// TIA Portal V20 export
// export: Created 2025-12-01T14:57:41.1647869Z, ExportSetting None, DisplayName Totally Integrated Automation Portal, DisplayVersion V20 Update 3, DisplayName TIA Portal Openness, DisplayVersion V20 Update 3, DisplayName TIA Portal Version Control Interface, DisplayVersion V20 Update 3, DisplayName STEP 7 Professional, DisplayVersion V20 Update 3, DisplayName STEP 7 Safety, DisplayVersion V20 Update 2, DisplayName WinCC Basic/Comfort/Advanced, DisplayVersion V20 Update 3, DisplayName WinCC Professional, DisplayVersion V20 Update 3, DisplayName WinCC Unified, DisplayVersion V20 Update 3
FUNCTION_BLOCK "FB384_Enfardadora_Paletizador_NDD"   // FB384, LAD
{ S7_Optimized_Access := 'FALSE' }
// stored: AutoNumber false, SetENOAutomatically false
   VAR_INPUT
      EstadoZona : "EstadoZona";
      NDB_Enfardadora : UInt;
      NumMaquina : UInt;
      PosicionActual : Int;
      DesHabitar_Enfa : Bool;
      PorCapas_Enfa : Bool;
      CheckElev_EnEnfardadora : Bool;
   END_VAR
   VAR
      MemoPosicionActual : Int;
      PosicionEnfardado : Int;
      VelocidadEnfardado : Int;
      ProgramaEnfardado : Int;
      PosEnfardadora_OK : Bool;
      PeticionSubirELEV : Bool;
      PeticionBajarELEV : Bool;
      EnPosEnfardado : Bool;
      DebajoPosEnfardado : Bool;
      EnPaletizadoUT : Bool;
      FinPaletizadoUT : Bool;
      SinEnfardadoUT { ExternalVisible := 'False'} : Bool;
      ConEnfardadoUT { ExternalVisible := 'False'} : Bool;
      IniciarEnfardado : Bool;
      FinEnfardado : Bool;
      ErrorEnfardado : Bool;
      RealizaCapaUT : Bool;
      HaciendoCapas : Bool;
      EnCicloEnfardado : Bool;
      EnCicloCapas : Bool;
      Elev_Subiendo : Bool;
      Elev_Bajando : Bool;
      ENFA_ET00 : Bool;
      ENFA_ET01 : Bool;
      ENFA_ET10 : Bool;
      ENFA_ET11 : Bool;
      ENFA_ET20 : Bool;
      ENFA_ET21 : Bool;
      ENFA_ET02 : Bool;
      ENFA_ET50 : Bool;
      ENFA_ET51 { ExternalVisible := 'False'} : Bool;
      t_march_enfa { S7_SetPoint := 'True'} : CTD_INT;
   END_VAR
   VAR_TEMP
      Entradas : "NDD_Enfardadora_Input";
      Salidas : "NDD_Enfardadora_Output";
      Guardar_AR1 : DWord;
      Guardar_AR2 : DWord;
      DB_Enfardadora : Word;
      P_Entradas : DWord;
      P_Salidas : DWord;
      P_Temporal : DWord;
      Margen : Int;
      AuxPosMax : Int;
      AuxPosMin : Int;
      Maquina : Word;
      DB_ColasMesas : Word;
      DB_DatosUT : Word;
      NumeroUT : UInt;
      SiguienteUT : UInt;
      MesaActual : UInt;
      MesaDestino : UInt;
      SinUT : Bool;
      AuxEstados : Bool;
   END_VAR
BEGIN

REGION Network 1: Inicializacion
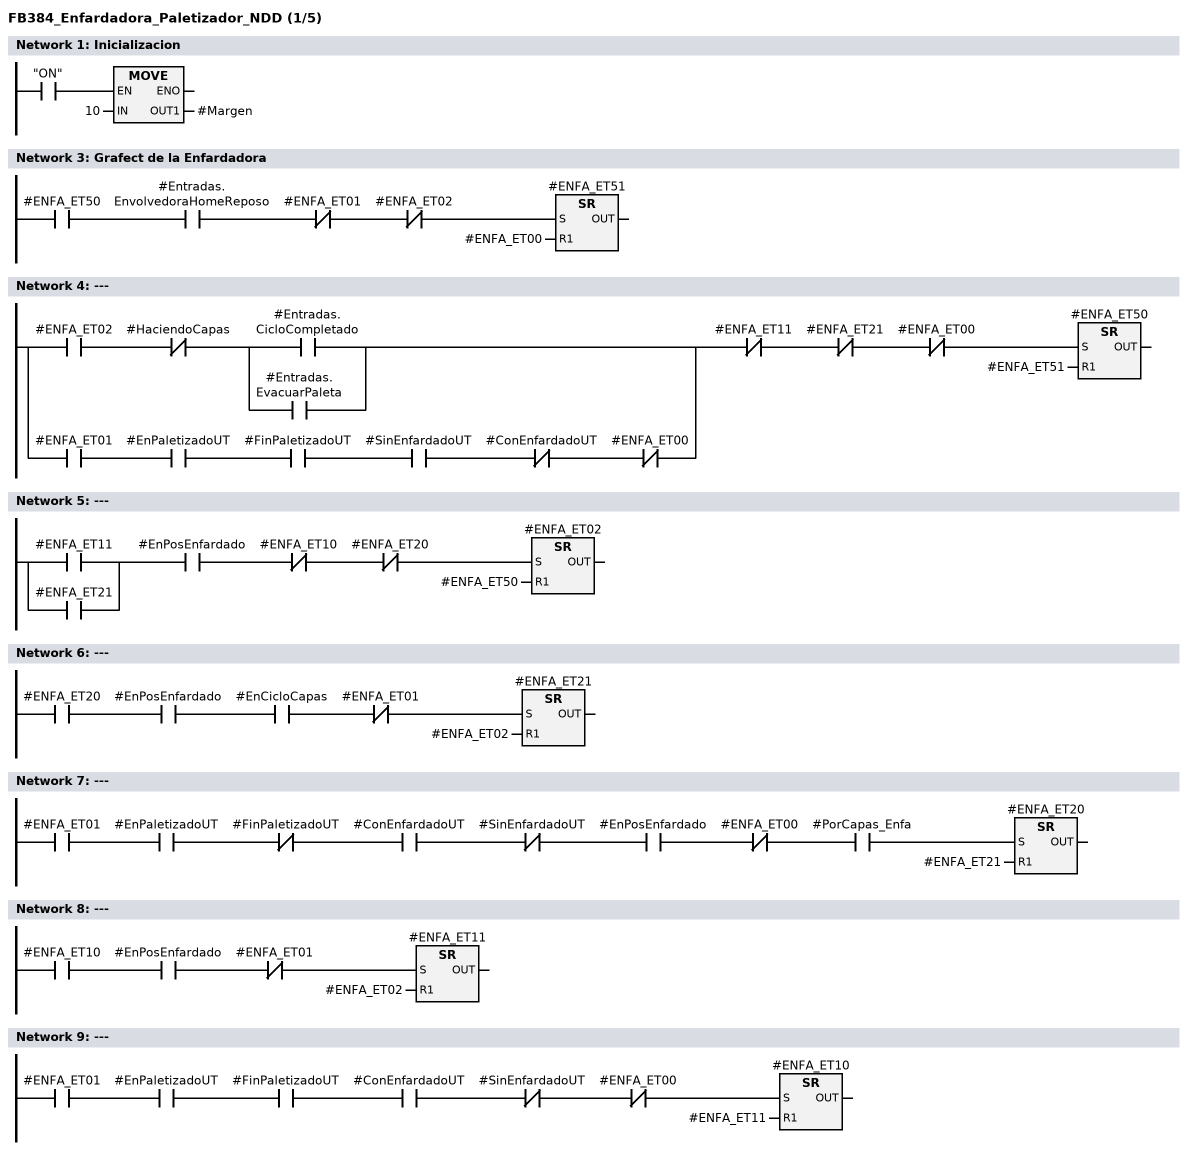
   RUNG wire#powerrail
      Contact( "ON" )
      { S7_GenerateENO := "TRUE" } Move(in := 10, out1 => #Margen)
   END_RUNG
   // the same network as SCL:
   IF "ON" THEN #Margen := 10; END_IF;
END_REGION

NETWORK
TITLE = Lectura de Datos
/////////////////////////////////////////////////////////////////////
/////////////////////////////////////////////////////////////////////
// - Inicializaciones Previas

      TAR1  #Guardar_AR1;  // - Guardar el AR1

      L     #NumMaquina;  // - Numero de Maquina
      T     #Maquina;

      L     #NDB_Enfardadora;  // - Numero de DB de Interlock
      T     #DB_Enfardadora;

/////////////////////////////////////////////////////////////////////
// -- Leer las entradas y salidas de la Enfardadora

      L     P##Entradas;  // --- Leer las Entradas
      T     #P_Entradas;
      L     P#0.0;
      T     #P_Temporal;

      OPN   DB [#DB_Enfardadora];  // - Bits de la Enfardadora
      L     DBD [#P_Temporal];
      T     LD [#P_Entradas];

      L     P#4.0;
      T     #P_Temporal;
      OPN   DB [#DB_Enfardadora];  // - Velocidad de Enfaradado
      L     DBW [#P_Temporal];
      T     #Entradas.VelocidadElevador;

      L     P#6.0;
      T     #P_Temporal;
      OPN   DB [#DB_Enfardadora];  // - Altura de Inicio de Enfardado
      L     DBW [#P_Temporal];
      T     #Entradas.AlturaInicioEnfardado;

      L     0;
      T     #Entradas.Libre_Int_08;

      L     P##Salidas;  // --- Leer las Salidas
      T     #P_Salidas;
      L     P#10.0;
      T     #P_Temporal;

      OPN   DB [#DB_Enfardadora];  // --- Bits
      L     DBD [#P_Temporal];
      T     LD [#P_Salidas];

      L     P#14.0;
      T     #P_Temporal;
      OPN   DB [#DB_Enfardadora];  // - Altura de la Paleta
      L     DBW [#P_Temporal];
      T     #Salidas.AlturaPaleta;

      L     P#16.0;
      T     #P_Temporal;
      OPN   DB [#DB_Enfardadora];  // - Posicion del Elevador
      L     DBW [#P_Temporal];
      T     #Salidas.AlturaElevador;

      L     P#18.0;
      T     #P_Temporal;
      OPN   DB [#DB_Enfardadora];  // - Programa
      L     DBW [#P_Temporal];
      T     #Salidas.Programa;


/////////////////////////////////////////////////////////////////////
/////////////////////////////////////////////////////////////////////
//  - Finalizacion

      LAR1  #Guardar_AR1;  // - Recuperar el AR1



REGION Network 3: Grafect de la Enfardadora
   RUNG wire#powerrail
      Contact( #ENFA_ET50 )
      Contact( #Entradas.EnvolvedoraHomeReposo )
      I_Contact( #ENFA_ET01 )
      I_Contact( #ENFA_ET02 )
      S_SR(operand := #ENFA_ET51, r1 := #ENFA_ET00)
   END_RUNG
   // the same network as SCL:
   IF #ENFA_ET50 AND #Entradas.EnvolvedoraHomeReposo AND NOT #ENFA_ET01 AND NOT #ENFA_ET02 THEN
       #ENFA_ET51 := TRUE;   // SR flip-flop
   END_IF;
   IF #ENFA_ET00 THEN #ENFA_ET51 := FALSE; END_IF;
END_REGION

REGION Network 4: ---
   RUNG wire#powerrail
      Contact( #ENFA_ET02 )
      I_Contact( #HaciendoCapas )
      wire#w1
      Contact( #Entradas.CicloCompletado )
      wire#w2
      I_Contact( #ENFA_ET11 )
      I_Contact( #ENFA_ET21 )
      I_Contact( #ENFA_ET00 )
      S_SR(operand := #ENFA_ET50, r1 := #ENFA_ET51)
   END_RUNG
   RUNG wire#w1
      Contact( #Entradas.EvacuarPaleta )
   END_RUNG wire#w2
   RUNG wire#powerrail
      Contact( #ENFA_ET01 )
      Contact( #EnPaletizadoUT )
      Contact( #FinPaletizadoUT )
      Contact( #SinEnfardadoUT )
      I_Contact( #ConEnfardadoUT )
      I_Contact( #ENFA_ET00 )
   END_RUNG wire#w2
   // the same network as SCL:
   IF ((#ENFA_ET02 AND NOT #HaciendoCapas AND (#Entradas.CicloCompletado OR #Entradas.EvacuarPaleta)) OR (#ENFA_ET01 AND #EnPaletizadoUT AND #FinPaletizadoUT AND #SinEnfardadoUT AND NOT #ConEnfardadoUT AND NOT #ENFA_ET00)) AND NOT #ENFA_ET11 AND NOT #ENFA_ET21 AND NOT #ENFA_ET00 THEN
       #ENFA_ET50 := TRUE;   // SR flip-flop
   END_IF;
   IF #ENFA_ET51 THEN #ENFA_ET50 := FALSE; END_IF;
END_REGION

REGION Network 5: ---
   RUNG wire#powerrail
      Contact( #ENFA_ET11 )
      wire#w1
      Contact( #EnPosEnfardado )
      I_Contact( #ENFA_ET10 )
      I_Contact( #ENFA_ET20 )
      S_SR(operand := #ENFA_ET02, r1 := #ENFA_ET50)
   END_RUNG
   RUNG wire#powerrail
      Contact( #ENFA_ET21 )
   END_RUNG wire#w1
   // the same network as SCL:
   IF (#ENFA_ET11 OR #ENFA_ET21) AND #EnPosEnfardado AND NOT #ENFA_ET10 AND NOT #ENFA_ET20 THEN
       #ENFA_ET02 := TRUE;   // SR flip-flop
   END_IF;
   IF #ENFA_ET50 THEN #ENFA_ET02 := FALSE; END_IF;
END_REGION

REGION Network 6: ---
   RUNG wire#powerrail
      Contact( #ENFA_ET20 )
      Contact( #EnPosEnfardado )
      Contact( #EnCicloCapas )
      I_Contact( #ENFA_ET01 )
      S_SR(operand := #ENFA_ET21, r1 := #ENFA_ET02)
   END_RUNG
   // the same network as SCL:
   IF #ENFA_ET20 AND #EnPosEnfardado AND #EnCicloCapas AND NOT #ENFA_ET01 THEN
       #ENFA_ET21 := TRUE;   // SR flip-flop
   END_IF;
   IF #ENFA_ET02 THEN #ENFA_ET21 := FALSE; END_IF;
END_REGION

REGION Network 7: ---
   RUNG wire#powerrail
      Contact( #ENFA_ET01 )
      Contact( #EnPaletizadoUT )
      I_Contact( #FinPaletizadoUT )
      Contact( #ConEnfardadoUT )
      I_Contact( #SinEnfardadoUT )
      Contact( #EnPosEnfardado )
      I_Contact( #ENFA_ET00 )
      Contact( #PorCapas_Enfa )
      S_SR(operand := #ENFA_ET20, r1 := #ENFA_ET21)
   END_RUNG
   // the same network as SCL:
   IF #ENFA_ET01 AND #EnPaletizadoUT AND NOT #FinPaletizadoUT AND #ConEnfardadoUT AND NOT #SinEnfardadoUT AND #EnPosEnfardado AND NOT #ENFA_ET00 AND #PorCapas_Enfa THEN
       #ENFA_ET20 := TRUE;   // SR flip-flop
   END_IF;
   IF #ENFA_ET21 THEN #ENFA_ET20 := FALSE; END_IF;
END_REGION

REGION Network 8: ---
   RUNG wire#powerrail
      Contact( #ENFA_ET10 )
      Contact( #EnPosEnfardado )
      I_Contact( #ENFA_ET01 )
      S_SR(operand := #ENFA_ET11, r1 := #ENFA_ET02)
   END_RUNG
   // the same network as SCL:
   IF #ENFA_ET10 AND #EnPosEnfardado AND NOT #ENFA_ET01 THEN
       #ENFA_ET11 := TRUE;   // SR flip-flop
   END_IF;
   IF #ENFA_ET02 THEN #ENFA_ET11 := FALSE; END_IF;
END_REGION

REGION Network 9: ---
   RUNG wire#powerrail
      Contact( #ENFA_ET01 )
      Contact( #EnPaletizadoUT )
      Contact( #FinPaletizadoUT )
      Contact( #ConEnfardadoUT )
      I_Contact( #SinEnfardadoUT )
      I_Contact( #ENFA_ET00 )
      S_SR(operand := #ENFA_ET10, r1 := #ENFA_ET11)
   END_RUNG
   // the same network as SCL:
   IF #ENFA_ET01 AND #EnPaletizadoUT AND #FinPaletizadoUT AND #ConEnfardadoUT AND NOT #SinEnfardadoUT AND NOT #ENFA_ET00 THEN
       #ENFA_ET10 := TRUE;   // SR flip-flop
   END_IF;
   IF #ENFA_ET11 THEN #ENFA_ET10 := FALSE; END_IF;
END_REGION

REGION Network 10: ---
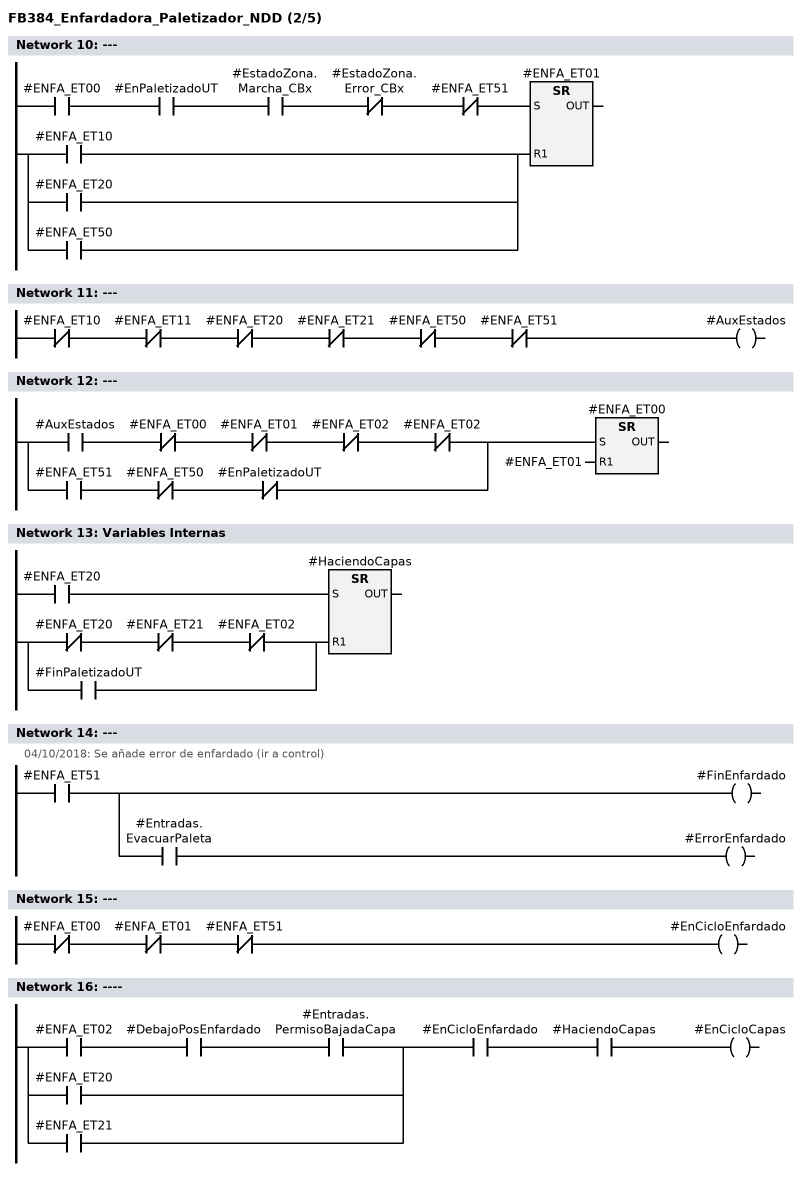
   RUNG wire#powerrail
      Contact( #ENFA_ET00 )
      Contact( #EnPaletizadoUT )
      Contact( #EstadoZona.Marcha_CBx )
      I_Contact( #EstadoZona.Error_CBx )
      I_Contact( #ENFA_ET51 )
      S_SR(operand := #ENFA_ET01, r1 := wire#w1)
   END_RUNG
   RUNG wire#powerrail
      Contact( #ENFA_ET10 )
   END_RUNG wire#w1
   RUNG wire#powerrail
      Contact( #ENFA_ET20 )
   END_RUNG wire#w1
   RUNG wire#powerrail
      Contact( #ENFA_ET50 )
   END_RUNG wire#w1
   // the same network as SCL:
   IF #ENFA_ET00 AND #EnPaletizadoUT AND #EstadoZona.Marcha_CBx AND NOT #EstadoZona.Error_CBx AND NOT #ENFA_ET51 THEN
       #ENFA_ET01 := TRUE;   // SR flip-flop
   END_IF;
   IF #ENFA_ET10 OR #ENFA_ET20 OR #ENFA_ET50 THEN #ENFA_ET01 := FALSE; END_IF;
END_REGION

REGION Network 11: ---
   RUNG wire#powerrail
      I_Contact( #ENFA_ET10 )
      I_Contact( #ENFA_ET11 )
      I_Contact( #ENFA_ET20 )
      I_Contact( #ENFA_ET21 )
      I_Contact( #ENFA_ET50 )
      I_Contact( #ENFA_ET51 )
      Coil( #AuxEstados )
   END_RUNG
   // the same network as SCL:
   #AuxEstados := NOT #ENFA_ET10 AND NOT #ENFA_ET11 AND NOT #ENFA_ET20 AND NOT #ENFA_ET21 AND NOT #ENFA_ET50 AND NOT #ENFA_ET51;
END_REGION

REGION Network 12: ---
   RUNG wire#powerrail
      Contact( #AuxEstados )
      I_Contact( #ENFA_ET00 )
      I_Contact( #ENFA_ET01 )
      I_Contact( #ENFA_ET02 )
      I_Contact( #ENFA_ET02 )
      wire#w1
      S_SR(operand := #ENFA_ET00, r1 := #ENFA_ET01)
   END_RUNG
   RUNG wire#powerrail
      Contact( #ENFA_ET51 )
      I_Contact( #ENFA_ET50 )
      I_Contact( #EnPaletizadoUT )
   END_RUNG wire#w1
   // the same network as SCL:
   IF (#AuxEstados AND NOT #ENFA_ET00 AND NOT #ENFA_ET01 AND NOT #ENFA_ET02 AND NOT #ENFA_ET02) OR (#ENFA_ET51 AND NOT #ENFA_ET50 AND NOT #EnPaletizadoUT) THEN
       #ENFA_ET00 := TRUE;   // SR flip-flop
   END_IF;
   IF #ENFA_ET01 THEN #ENFA_ET00 := FALSE; END_IF;
END_REGION

REGION Network 13: Variables Internas
   RUNG wire#powerrail
      Contact( #ENFA_ET20 )
      S_SR(operand := #HaciendoCapas, r1 := wire#w1)
   END_RUNG
   RUNG wire#powerrail
      I_Contact( #ENFA_ET20 )
      I_Contact( #ENFA_ET21 )
      I_Contact( #ENFA_ET02 )
   END_RUNG wire#w1
   RUNG wire#powerrail
      Contact( #FinPaletizadoUT )
   END_RUNG wire#w1
   // the same network as SCL:
   IF #ENFA_ET20 THEN
       #HaciendoCapas := TRUE;   // SR flip-flop
   END_IF;
   IF (NOT #ENFA_ET20 AND NOT #ENFA_ET21 AND NOT #ENFA_ET02) OR #FinPaletizadoUT THEN
       #HaciendoCapas := FALSE;
   END_IF;
END_REGION

REGION Network 14: ---
   // 04/10/2018: Se añade error de enfardado (ir a control)
   RUNG wire#powerrail
      Contact( #ENFA_ET51 )
      wire#w1
      Coil( #FinEnfardado )
   END_RUNG
   RUNG wire#w1
      Contact( #Entradas.EvacuarPaleta )
      Coil( #ErrorEnfardado )
   END_RUNG
   // the same network as SCL:
   #FinEnfardado := #ENFA_ET51;
   #ErrorEnfardado := #ENFA_ET51 AND #Entradas.EvacuarPaleta;
END_REGION

REGION Network 15: ---
   RUNG wire#powerrail
      I_Contact( #ENFA_ET00 )
      I_Contact( #ENFA_ET01 )
      I_Contact( #ENFA_ET51 )
      Coil( #EnCicloEnfardado )
   END_RUNG
   // the same network as SCL:
   #EnCicloEnfardado := NOT #ENFA_ET00 AND NOT #ENFA_ET01 AND NOT #ENFA_ET51;
END_REGION

REGION Network 16: ----
   RUNG wire#powerrail
      Contact( #ENFA_ET02 )
      Contact( #DebajoPosEnfardado )
      Contact( #Entradas.PermisoBajadaCapa )
      wire#w1
      Contact( #EnCicloEnfardado )
      Contact( #HaciendoCapas )
      Coil( #EnCicloCapas )
   END_RUNG
   RUNG wire#powerrail
      Contact( #ENFA_ET20 )
   END_RUNG wire#w1
   RUNG wire#powerrail
      Contact( #ENFA_ET21 )
   END_RUNG wire#w1
   // the same network as SCL:
   #EnCicloCapas := ((#ENFA_ET02 AND #DebajoPosEnfardado AND #Entradas.PermisoBajadaCapa) OR #ENFA_ET20 OR #ENFA_ET21) AND #EnCicloEnfardado AND #HaciendoCapas;
END_REGION

REGION Network 17: ---
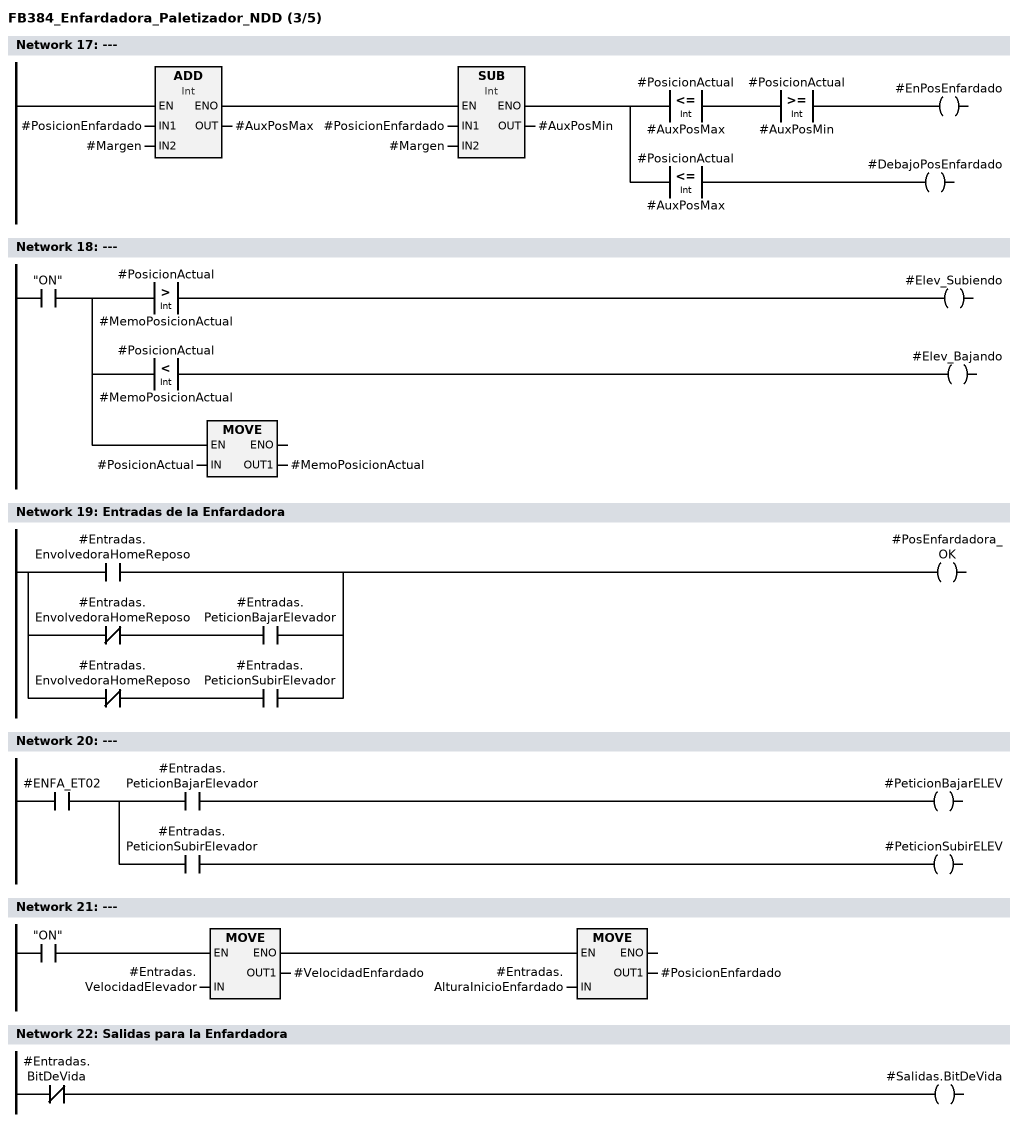
   RUNG wire#powerrail
      { S7_Templates := "SrcType := Int"; S7_GenerateENO := "TRUE" } Add(in1 := #PosicionEnfardado, in2 := #Margen, out => #AuxPosMax)
      { S7_Templates := "SrcType := Int"; S7_GenerateENO := "TRUE" } Sub(in1 := #PosicionEnfardado, in2 := #Margen, out => #AuxPosMin)
      wire#w1
      { S7_Templates := "SrcType := Int" } LE_Contact(in1 := #PosicionActual, in2 := #AuxPosMax)
      { S7_Templates := "SrcType := Int" } GE_Contact(in1 := #PosicionActual, in2 := #AuxPosMin)
      Coil( #EnPosEnfardado )
   END_RUNG
   RUNG wire#w1
      { S7_Templates := "SrcType := Int" } LE_Contact(in1 := #PosicionActual, in2 := #AuxPosMax)
      Coil( #DebajoPosEnfardado )
   END_RUNG
   // the same network as SCL:
   // ENO of a box is taken as its EN; it also drops when the box reports an error
   #AuxPosMax := #PosicionEnfardado + #Margen;
   #AuxPosMin := #PosicionEnfardado - #Margen;
   #EnPosEnfardado := (#PosicionActual <= #AuxPosMax) AND (#PosicionActual >= #AuxPosMin);
   #DebajoPosEnfardado := #PosicionActual <= #AuxPosMax;
END_REGION

REGION Network 18: ---
   RUNG wire#powerrail
      Contact( "ON" )
      wire#w1
      { S7_Templates := "SrcType := Int" } GT_Contact(in1 := #PosicionActual, in2 := #MemoPosicionActual)
      Coil( #Elev_Subiendo )
   END_RUNG
   RUNG wire#w1
      { S7_Templates := "SrcType := Int" } LT_Contact(in1 := #PosicionActual, in2 := #MemoPosicionActual)
      Coil( #Elev_Bajando )
   END_RUNG
   RUNG wire#w1
      { S7_GenerateENO := "TRUE" } Move(in := #PosicionActual, out1 => #MemoPosicionActual)
   END_RUNG
   // the same network as SCL:
   #Elev_Subiendo := "ON" AND (#PosicionActual > #MemoPosicionActual);
   #Elev_Bajando := "ON" AND (#PosicionActual < #MemoPosicionActual);
   IF "ON" THEN #MemoPosicionActual := #PosicionActual; END_IF;
END_REGION

REGION Network 19: Entradas de la Enfardadora
   RUNG wire#powerrail
      Contact( #Entradas.EnvolvedoraHomeReposo )
      wire#w1
      Coil( #PosEnfardadora_OK )
   END_RUNG
   RUNG wire#powerrail
      I_Contact( #Entradas.EnvolvedoraHomeReposo )
      Contact( #Entradas.PeticionBajarElevador )
   END_RUNG wire#w1
   RUNG wire#powerrail
      I_Contact( #Entradas.EnvolvedoraHomeReposo )
      Contact( #Entradas.PeticionSubirElevador )
   END_RUNG wire#w1
   // the same network as SCL:
   #PosEnfardadora_OK := #Entradas.EnvolvedoraHomeReposo OR (NOT #Entradas.EnvolvedoraHomeReposo AND #Entradas.PeticionBajarElevador) OR (NOT #Entradas.EnvolvedoraHomeReposo AND #Entradas.PeticionSubirElevador);
END_REGION

REGION Network 20: ---
   RUNG wire#powerrail
      Contact( #ENFA_ET02 )
      wire#w1
      Contact( #Entradas.PeticionBajarElevador )
      Coil( #PeticionBajarELEV )
   END_RUNG
   RUNG wire#w1
      Contact( #Entradas.PeticionSubirElevador )
      Coil( #PeticionSubirELEV )
   END_RUNG
   // the same network as SCL:
   #PeticionBajarELEV := #ENFA_ET02 AND #Entradas.PeticionBajarElevador;
   #PeticionSubirELEV := #ENFA_ET02 AND #Entradas.PeticionSubirElevador;
END_REGION

REGION Network 21: ---
   RUNG wire#powerrail
      Contact( "ON" )
      { S7_GenerateENO := "TRUE" } Move(in := #Entradas.VelocidadElevador, out1 => #VelocidadEnfardado)
      { S7_GenerateENO := "TRUE" } Move(in := #Entradas.AlturaInicioEnfardado, out1 => #PosicionEnfardado)
   END_RUNG
   // the same network as SCL:
   // ENO of a box is taken as its EN; it also drops when the box reports an error
   IF "ON" THEN
       #VelocidadEnfardado := #Entradas.VelocidadElevador;
       #PosicionEnfardado := #Entradas.AlturaInicioEnfardado;
   END_IF;
END_REGION

REGION Network 22: Salidas para la Enfardadora
   RUNG wire#powerrail
      I_Contact( #Entradas.BitDeVida )
      Coil( #Salidas.BitDeVida )
   END_RUNG
   // the same network as SCL:
   #Salidas.BitDeVida := NOT #Entradas.BitDeVida;
END_REGION

REGION Network 23: ---
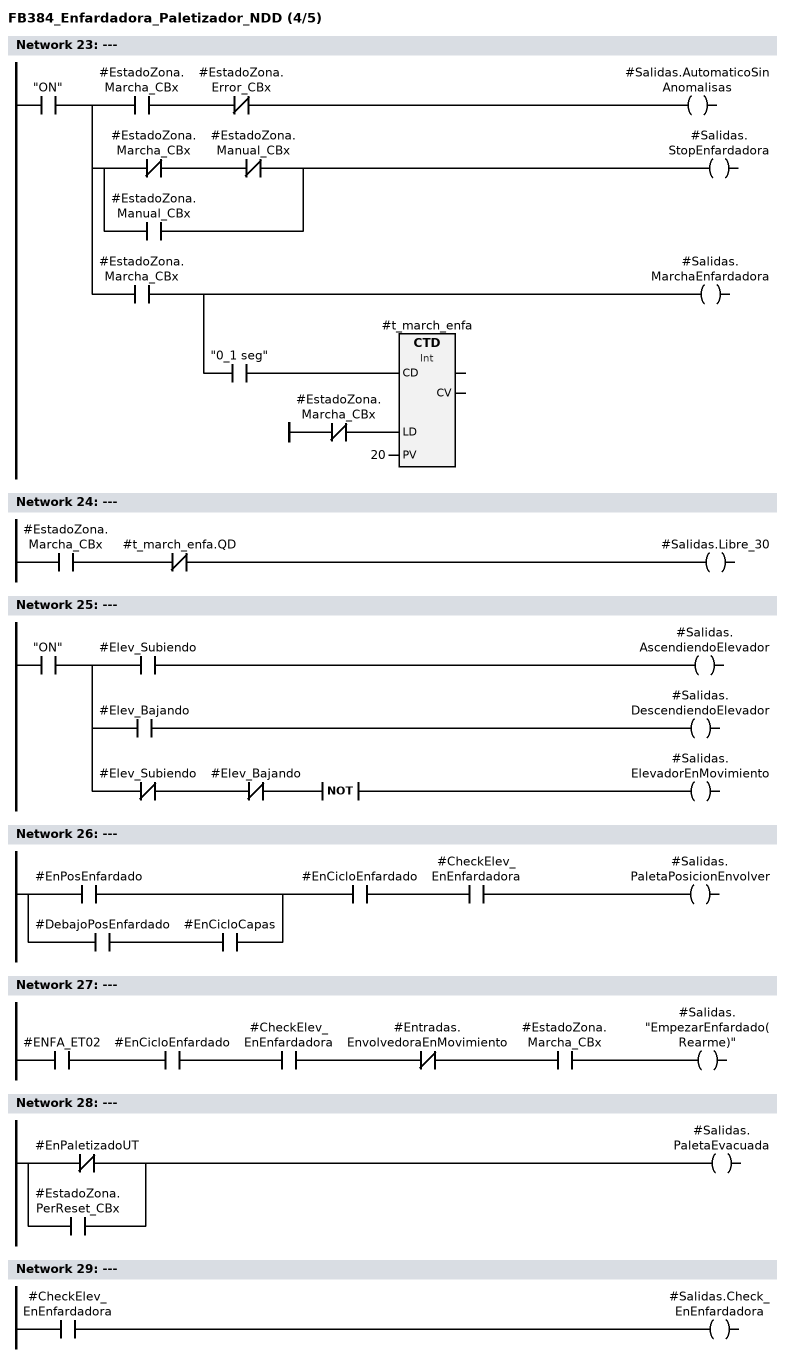
   RUNG wire#powerrail
      Contact( "ON" )
      wire#w1
      Contact( #EstadoZona.Marcha_CBx )
      I_Contact( #EstadoZona.Error_CBx )
      Coil( #Salidas.AutomaticoSinAnomalisas )
   END_RUNG
   RUNG wire#w1
      I_Contact( #EstadoZona.Marcha_CBx )
      I_Contact( #EstadoZona.Manual_CBx )
      wire#w2
      Coil( #Salidas.StopEnfardadora )
   END_RUNG
   RUNG wire#w1
      Contact( #EstadoZona.Manual_CBx )
   END_RUNG wire#w2
   RUNG wire#w1
      Contact( #EstadoZona.Marcha_CBx )
      wire#w3
      Coil( #Salidas.MarchaEnfardadora )
   END_RUNG
   RUNG wire#w3
      Contact( "0_1 seg" )
      { S7_Templates := "value_type := Int" } #t_march_enfa.CTD(ld := wire#w4, pv := 20, cv =>)
   END_RUNG
   RUNG wire#powerrail
      I_Contact( #EstadoZona.Marcha_CBx )
   END_RUNG wire#w4
   // the same network as SCL:
   #Salidas.AutomaticoSinAnomalisas := "ON" AND #EstadoZona.Marcha_CBx AND NOT #EstadoZona.Error_CBx;
   #Salidas.StopEnfardadora := "ON" AND ((NOT #EstadoZona.Marcha_CBx AND NOT #EstadoZona.Manual_CBx) OR #EstadoZona.Manual_CBx);
   #Salidas.MarchaEnfardadora := "ON" AND #EstadoZona.Marcha_CBx;
   #t_march_enfa(CD := #Salidas.MarchaEnfardadora AND "0_1 seg", LD := NOT #EstadoZona.Marcha_CBx, PV := 20);   // CTD
END_REGION

REGION Network 24: ---
   RUNG wire#powerrail
      Contact( #EstadoZona.Marcha_CBx )
      I_Contact( #t_march_enfa.QD )
      Coil( #Salidas.Libre_30 )
   END_RUNG
   // the same network as SCL:
   #Salidas.Libre_30 := #EstadoZona.Marcha_CBx AND NOT #t_march_enfa.QD;
END_REGION

REGION Network 25: ---
   RUNG wire#powerrail
      Contact( "ON" )
      wire#w1
      Contact( #Elev_Subiendo )
      Coil( #Salidas.AscendiendoElevador )
   END_RUNG
   RUNG wire#w1
      Contact( #Elev_Bajando )
      Coil( #Salidas.DescendiendoElevador )
   END_RUNG
   RUNG wire#w1
      I_Contact( #Elev_Subiendo )
      I_Contact( #Elev_Bajando )
      Not()
      Coil( #Salidas.ElevadorEnMovimiento )
   END_RUNG
   // the same network as SCL:
   #Salidas.AscendiendoElevador := "ON" AND #Elev_Subiendo;
   #Salidas.DescendiendoElevador := "ON" AND #Elev_Bajando;
   #Salidas.ElevadorEnMovimiento := NOT ("ON" AND NOT #Elev_Subiendo AND NOT #Elev_Bajando);
END_REGION

REGION Network 26: ---
   RUNG wire#powerrail
      Contact( #EnPosEnfardado )
      wire#w1
      Contact( #EnCicloEnfardado )
      Contact( #CheckElev_EnEnfardadora )
      Coil( #Salidas.PaletaPosicionEnvolver )
   END_RUNG
   RUNG wire#powerrail
      Contact( #DebajoPosEnfardado )
      Contact( #EnCicloCapas )
   END_RUNG wire#w1
   // the same network as SCL:
   #Salidas.PaletaPosicionEnvolver := (#EnPosEnfardado OR (#DebajoPosEnfardado AND #EnCicloCapas)) AND #EnCicloEnfardado AND #CheckElev_EnEnfardadora;
END_REGION

REGION Network 27: ---
   RUNG wire#powerrail
      Contact( #ENFA_ET02 )
      Contact( #EnCicloEnfardado )
      Contact( #CheckElev_EnEnfardadora )
      I_Contact( #Entradas.EnvolvedoraEnMovimiento )
      Contact( #EstadoZona.Marcha_CBx )
      Coil( #Salidas."EmpezarEnfardado(Rearme)" )
   END_RUNG
   // the same network as SCL:
   #Salidas."EmpezarEnfardado(Rearme)" := #ENFA_ET02 AND #EnCicloEnfardado AND #CheckElev_EnEnfardadora AND NOT #Entradas.EnvolvedoraEnMovimiento AND #EstadoZona.Marcha_CBx;
END_REGION

REGION Network 28: ---
   RUNG wire#powerrail
      I_Contact( #EnPaletizadoUT )
      wire#w1
      Coil( #Salidas.PaletaEvacuada )
   END_RUNG
   RUNG wire#powerrail
      Contact( #EstadoZona.PerReset_CBx )
   END_RUNG wire#w1
   // the same network as SCL:
   #Salidas.PaletaEvacuada := NOT #EnPaletizadoUT OR #EstadoZona.PerReset_CBx;
END_REGION

REGION Network 29: ---
   RUNG wire#powerrail
      Contact( #CheckElev_EnEnfardadora )
      Coil( #Salidas.Check_EnEnfardadora )
   END_RUNG
   // the same network as SCL:
   #Salidas.Check_EnEnfardadora := #CheckElev_EnEnfardadora;
END_REGION

REGION Network 30: ---
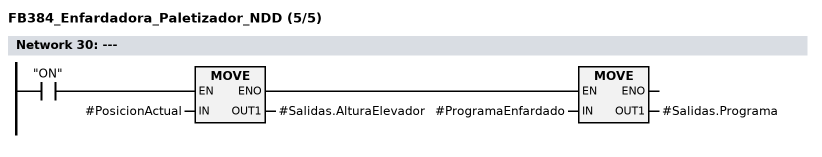
   RUNG wire#powerrail
      Contact( "ON" )
      { S7_GenerateENO := "TRUE" } Move(in := #PosicionActual, out1 => #Salidas.AlturaElevador)
      { S7_GenerateENO := "TRUE" } Move(in := #ProgramaEnfardado, out1 => #Salidas.Programa)
   END_RUNG
   // the same network as SCL:
   // ENO of a box is taken as its EN; it also drops when the box reports an error
   IF "ON" THEN
       #Salidas.AlturaElevador := #PosicionActual;
       #Salidas.Programa := #ProgramaEnfardado;
   END_IF;
END_REGION

NETWORK
TITLE = Escritura de Datos
/////////////////////////////////////////////////////////////////////
/////////////////////////////////////////////////////////////////////
// - Inicializaciones Previas

      TAR1  #Guardar_AR1;  // - Guardar el AR1


/////////////////////////////////////////////////////////////////////
// -- Escribir las salidas de la Enfardadora

      L     P##Salidas;  // --- Escribir las Salidas
      T     #P_Salidas;
      L     P#10.0;
      T     #P_Temporal;

      OPN   DB [#DB_Enfardadora];  // - Bits
      L     LD [#P_Salidas];
      T     DBD [#P_Temporal];

      L     P#14.0;
      T     #P_Temporal;
      OPN   DB [#DB_Enfardadora];  // - Altura de la  Paleta
      L     #Salidas.AlturaPaleta;
      T     DBW [#P_Temporal];

      L     P#16.0;
      T     #P_Temporal;
      OPN   DB [#DB_Enfardadora];  // - Posicion del Elevador
      L     #Salidas.AlturaElevador;
      T     DBW [#P_Temporal];

      L     P#18.0;
      T     #P_Temporal;
      OPN   DB [#DB_Enfardadora];  // - Programa
      L     #Salidas.Programa;
      T     DBW [#P_Temporal];


/////////////////////////////////////////////////////////////////////
/////////////////////////////////////////////////////////////////////
//  - Finalizacion

      LAR1  #Guardar_AR1;  // - Recuperar el AR1


END_FUNCTION_BLOCK
